(* IEC 61131-3 sources: esstee/src/tests/programs/loops, 7 files *)

(* ---- for.ST ---- *)
PROGRAM t

VAR
	itr : INT;
	out : ARRAY[1..5] of INT;
	out2 : ARRAY[1..5] of INT;
END_VAR

for itr := 1 to 5 do
    out[itr] := itr;
    out2[itr] := itr * 2;
end_for;

END_PROGRAM

(* ---- forexit.ST ---- *)
PROGRAM t

VAR
	itr : INT;
	out : ARRAY[1..5] of INT;
END_VAR

for itr := 1 to 5 do
    out[itr] := itr;

    if itr = 2 then
       exit;
    end_if;

end_for;

END_PROGRAM

(* ---- forrange.ST ---- *)
PROGRAM t

VAR
	from_value : INT;
	to_value : INT;
	itr : INT;
	sum : INT;
END_VAR

for itr := from_value to to_value do
    sum := sum + itr;
end_for;

END_PROGRAM

(* ---- repeat.ST ---- *)
PROGRAM t

VAR
	itr : INT := 0;
	control : INT := 0;
	control_two : INT := 0;
	itr_two : INT := 0;
END_VAR

repeat
      itr := itr + 1;

      if itr > 5 then
      	 exit;
      end_if;

      control := control + 1;
until False
end_repeat;

repeat
      control_two := control_two + 1;
until True
end_repeat;

repeat
	itr_two := itr_two + 1;
until itr_two > 4
end_repeat;

END_PROGRAM

(* ---- repeatnotbool.ST ---- *)
PROGRAM t

VAR
	itr : INT := 0;
END_VAR

repeat
      itr := itr + 1;
until itr
end_repeat;

END_PROGRAM

(* ---- while.ST ---- *)
PROGRAM t

VAR
	itr : INT := 0;
	control : INT := 0;
	control_two : INT := 0;
	itr_two : INT := 0;
END_VAR

while True do
      itr := itr + 1;

      if itr > 5 then
      	 exit;
      end_if;

      control := control + 1;

end_while;

while False do
      control_two := 100;
end_while;

while itr_two < 4 do
      itr_two := itr_two + 1;
end_while;

END_PROGRAM

(* ---- whilenotbool.ST ---- *)
PROGRAM t

VAR
	itr : INT := 0;
END_VAR

while itr do
      itr := itr + 1;
end_while;

END_PROGRAM
